PROGRAM MAIN
VAR
	bChangeSeparatorToComma: BOOL;
END_VAR

IF bChangeSeparatorToComma THEN
	DEFAULT_CSV_FIELD_SEP := 16#2C;(* Comma ASCII code *)
ELSE
	DEFAULT_CSV_FIELD_SEP := 16#3B;(* Semicolon ASCII code *)
END_IF



	//ReadCSV();
	
	ReadCSVSecondPractice();

END_PROGRAM

(* stored: Version 1.1.0.1, ProductVersion 3.1.4022.16
   POU MAIN: Id {534ab4b7-690d-4c49-9055-9f6244e09a5e}, SpecialFunc None *)
